{attribute 'GeneratedUsingTerminal: EK1100-0000-0018'}
{attribute addProperty BoxType "EK1100-0000-0018"}
{attribute addProperty Id "Beckhoff_EP8xxxEK1122Beckhoff_EP8xxxEK1122_7348582A282"}
{attribute addProperty CRC "2143852275"}
{attribute addProperty Size "282"}
{attribute addProperty Name "Beckhoff EP8xxx"}
TYPE Beckhoff_EP8xxx_7FC896F3 EXTENDS EK1100_1FC0878B :
STRUCT
	{attribute addProperty Name "Beckhoff EP8xxxEK1122"}
	{attribute addProperty PreviousPort "Beckhoff EP8xxx : B"}
	Beckhoff_EP8xxxEK1122 : Beckhoff_EP8xxxEK1122_7348582A;
END_STRUCT
END_TYPE

(* stored: Version 1.2.0.0, ProductVersion 3.1.4024.11
   DUT Beckhoff_EP8xxx_7FC896F3: Id {6e07d135-fdaf-4a37-9988-c7b1b9be4d75} *)
